FUNCTION_BLOCK T_TestEvent_UsesEventArgs EXTENDS T_EventBase 
VAR
    Handler : I_TestEventHandler_UsesEventArgs;
END_VAR

METHOD PRIVATE CallHandler
VAR_INPUT
    HandlerBase : I_EventHandlerBase;
    EventArgs   : I_StreamReader;
END_VAR
IF __QUERYINTERFACE(HandlerBase,Handler) THEN
    Handler.OnThisEvent(EventArgs);
//ELSE
//    tcl_BaseClasses.F_LogError('Event Handling',F_FormatStringEx1('Error raising %s - invalid handler',EventName));
END_IF
END_METHOD

METHOD IsHandlerSupported : BOOL
VAR_INPUT
    HandlerBase : I_EventHandlerBase;
END_VAR
IF __QUERYINTERFACE(HandlerBase,Handler) THEN
    IsHandlerSupported := TRUE;
END_IF
END_METHOD

END_FUNCTION_BLOCK

(* stored: Version 1.1.0.1, ProductVersion 3.1.4024.4
   POU T_TestEvent_UsesEventArgs: Id {53484359-1014-40a2-861a-ebe4d2e6097c}, SpecialFunc None
   Method CallHandler: Id {f160dfaf-006a-40a9-a062-4ad03f8b1f56}
   Method IsHandlerSupported: Id {246727ba-99c5-40b5-aa38-8d43578f023b} *)
